// ---- FBs/Setpoint Optimizer/FB_SPOpt_HybridAirSystem.TcPOU
{attribute 'hide_all_locals'}
FUNCTION_BLOCK FB_SPOpt_HybridAirSystem
VAR_INPUT PERSISTENT
	bEnable							: BOOL;									//Enable or dissable thsi Function
END_VAR
VAR_INPUT
	byStateSystemIn					: BYTE;									//Actual State from the System. 0 = off, 1 = Heating mode on, 2 = Cooling Mode on
	rFlowAirTempIn					: REAL;									//Actual Flow Air Temperature
	rReturnAirTempIn				: REAL;									//Actual Return Air Temperature
	rInToOutAirTempIn				: REAL;									//Actual outdoor air flow temperature
	rOutToInAirTempIn				: REAL;									//Actual indoor air flow temperature
END_VAR
VAR_OUTPUT
	bError							: BOOL;									//Error from this Fuction
	byStateSystemOut				: BYTE;									//{#lynus.ag#()} //State from the System. 0 = off, 1 = Heating mode on, 2 = Cooling Mode on		
	rFlowAirTempOut					: REAL;									//{#lynus.ag#()} //Flow Air Temperature to send to the Backend Service.
	rReturnAirTempOut				: REAL;									//{#lynus.ag#()} //Return Air Temperature to send to the Backend Service.
	rInToOutAirTempOut				: REAL;									//{#lynus.ag#()} //Outdoor air flow temperature to send to the Backend Service.
	rOutToInAirTempOut				: REAL;									//{#lynus.ag#()} //Indoor air flow temperature to send to the Backend Service.
	diNrOfSPOpt_OUT					: DINT;									//Active Number from Setpoint Optimizer for using on other functions
END_VAR
VAR
	fbNumberDevice					: FB_NumberOfDevice;					//Function block to calcualte the number of the Device
	timDissableFunctions			: TON;									//Timer to dissable the Function after Lynus_Standards.Constants_General.tTimeDissableLynusFunctions Days without connection to the Lynus Cloud
	timResetConnectionOnGVL			: TON;									//Timer to try reset the connection Flag on the GVL. (When somebody delete the Connection Function and make only a onlinechange)
END_VAR

//Creator : Kai Ebensperger
//Company : Lynus AG
//Date : 03.12.2021
//Version : 1.0.0.0

//This Function is a Help Function for the Setpoint Optimizer on our Backend System
//Here we can read in the neccessary Values for a Hybrid Air System from a external Service and can send then to the Backend System for optimizing
//Hybrid System can bee heating and cooling
//Its Helpfull if we work with the TMC File

(*----------------------------------------------------------------------------------------Limits---------------------------------------------------------------------------------------------------------------*)

byStateSystemIn := LIMIT(0,byStateSystemIn,2);
	rFlowAirTempIn := LIMIT(-30,rFlowAirTempIn,150);
		rReturnAirTempIn := LIMIT(-30,rReturnAirTempIn,150);
			rInToOutAirTempIn := LIMIT(-30,rInToOutAirTempIn,150);
				rOutToInAirTempIn := LIMIT(-30,rOutToInAirTempIn,150);

(*-------------------------------------------------------------Calcualte the number of SP Opttimizer---------------------------------------------------------------*)

fbNumberDevice(
	diActualNumberOfDevices:= Lynus_Standards.GVL_Energy.stNumberOfDevices.diNumberOfSetPointOpt, 
	diMaxNumberOfDevices:= Constants_Energy.diMaxNumberOfSetPointOpt, 
	udiCounterOnlineChange:= TwinCAT_SystemInfoVarList._AppInfo.OnlineChangeCnt, 
	bNumberIsCalculatet=> , 
	bFPNumberIsCalculatet=> , 
	bOnlineChange=> , 
	diNumberForThisDevice=> diNrOfSPOpt_OUT, 
	diNumberOfTotalDevices=> );

//Write new Numer on GVL
IF fbNumberDevice.bFPNumberIsCalculatet THEN
	Lynus_Standards.GVL_Energy.stNumberOfDevices.diNumberOfSetPointOpt := fbNumberDevice.diNumberOfTotalDevices;	
END_IF 

//Delete old Number on GVL
IF fbNumberDevice.bOnlineChange THEN 
	Lynus_Standards.GVL_Energy.stNumberOfDevices.diNumberOfSetPointOpt := diNrOfSPOpt_OUT;
END_IF								
				
(*-------------------------------------------------------------Service from Backend is ready and check the connection to backen for dissabel/enable EMS Function---------------------------------------------------------------*)

//Try to reset the variable for connection on the GVL. When all is normal then the Lynus Mqtt connection function set this variable to true in the next cycle
//When we have no connection to the backend or no HB from the Service then after Lynus_Standards.Constants_General.tTimeDissableLynusFunctions days the EMS is dissabled with all of his functionalities
timResetConnectionOnGVL(IN:= NOT timResetConnectionOnGVL.Q, PT:= T#1H, Q=> , ET=> );
	IF timResetConnectionOnGVL.Q THEN Lynus_Standards.GVL_Communicator.bStateConnectionToEnableFunctions := FALSE; END_IF
		IF NOT Lynus_Standards.GVL_Communicator.bStateConnectionToEnableFunctions THEN timDissableFunctions.IN := TRUE; ELSE timDissableFunctions.IN := FALSE; END_IF  
			timDissableFunctions(IN:= , PT:= Lynus_Standards.Constants_General.tTimeDissableLynusFunctions, Q=> , ET=> );

(*------------------------------------------------------------------Error----------------------------------------------------------------------------*)	

IF Lynus_Standards.GVL_Energy.stNumberOfDevices.diNumberOfSetPointOpt > Constants_Energy.diMaxNumberOfSetPointOpt THEN bError := TRUE; ELSE bError := FALSE; END_IF 			
			
(*-------------------------------------------------------------------------------------In to Out---------------------------------------------------------------------------------------*)

byStateSystemOut := byStateSystemIn;
	rFlowAirTempOut := rFlowAirTempIn;
		rReturnAirTempOut := rReturnAirTempIn;	
			rInToOutAirTempOut := rInToOutAirTempIn;
				rOutToInAirTempOut := rOutToInAirTempIn;		

IF NOT bEnable OR timDissableFunctions.Q OR Lynus_Standards.GVL_Energy.stNumberOfDevices.diNumberOfSetPointOpt > Constants_Energy.diMaxNumberOfSetPointOpt THEN
	byStateSystemOut := 0;	
END_IF

END_FUNCTION_BLOCK

// ---- FBs/Setpoint Optimizer/FB_SPOpt_HybridWaterSystem.TcPOU
{attribute 'hide_all_locals'}
FUNCTION_BLOCK FB_SPOpt_HybridWaterSystem
VAR_INPUT PERSISTENT
	bEnable							: BOOL;									//Enable or dissable thsi Function
END_VAR
VAR_INPUT
	byStateSystemIn					: BYTE;									//Actual State from the System. 0 = off, 1 = Heating mode on, 2 = Cooling Mode on
	rFlowTempIn						: REAL;									//Actual Flow Temperature
	rReturnTempIn					: REAL;									//Actual Return Temperature
END_VAR
VAR_OUTPUT
	bError							: BOOL;									//Error from this Fuction
	byStateSystemOut				: BYTE;									//{#lynus.ag#()} //State from the System. 0 = off, 1 = Heating mode on, 2 = Cooling Mode on	
	rFlowTempOut					: REAL;									//{#lynus.ag#()} //Flow Temperature to send to the Backend Service.
	rReturnTempOut					: REAL;									//{#lynus.ag#()} //Return Temperature to send to the Backend Service.
	diNrOfSPOpt_OUT					: DINT;									//Active Number from Setpoint Optimizer for using on other functions
END_VAR
VAR
	fbNumberDevice					: FB_NumberOfDevice;					//Function block to calcualte the number of the Device
	timDissableFunctions			: TON;									//Timer to dissable the Function after Lynus_Standards.Constants_General.tTimeDissableLynusFunctions Days without connection to the Lynus Cloud
	timResetConnectionOnGVL			: TON;									//Timer to try reset the connection Flag on the GVL. (When somebody delete the Connection Function and make only a onlinechange)
END_VAR

//Creator : Kai Ebensperger
//Company : Lynus AG
//Date : 03.12.2021
//Version : 1.0.0.0

//This Function is a Help Function for the Setpoint Optimizer on our Backend System
//Here we can read in the neccessary Values for a Hybrid Water System from a external Service and can send then to the Backend System for optimizing
//Hybrid System can bee heating and cooling
//Its Helpfull if we work with the TMC File

(*----------------------------------------------------------------------------------------Limits---------------------------------------------------------------------------------------------------------------*)

byStateSystemIn := LIMIT(0,byStateSystemIn,2);
	rFlowTempIn := LIMIT(-30,rFlowTempIn,180);
		rReturnTempIn := LIMIT(-30,rReturnTempIn,180);

(*-------------------------------------------------------------Calcualte the number of SP Opttimizer---------------------------------------------------------------*)

fbNumberDevice(
	diActualNumberOfDevices:= Lynus_Standards.GVL_Energy.stNumberOfDevices.diNumberOfSetPointOpt, 
	diMaxNumberOfDevices:= Constants_Energy.diMaxNumberOfSetPointOpt, 
	udiCounterOnlineChange:= TwinCAT_SystemInfoVarList._AppInfo.OnlineChangeCnt, 
	bNumberIsCalculatet=> , 
	bFPNumberIsCalculatet=> , 
	bOnlineChange=> , 
	diNumberForThisDevice=> diNrOfSPOpt_OUT, 
	diNumberOfTotalDevices=> );

//Write new Numer on GVL
IF fbNumberDevice.bFPNumberIsCalculatet THEN
	Lynus_Standards.GVL_Energy.stNumberOfDevices.diNumberOfSetPointOpt := fbNumberDevice.diNumberOfTotalDevices;	
END_IF 

//Delete old Number on GVL
IF fbNumberDevice.bOnlineChange THEN 
	Lynus_Standards.GVL_Energy.stNumberOfDevices.diNumberOfSetPointOpt := diNrOfSPOpt_OUT;
END_IF			
		
(*-------------------------------------------------------------Service from Backend is ready and check the connection to backen for dissabel/enable EMS Function---------------------------------------------------------------*)

//Try to reset the variable for connection on the GVL. When all is normal then the Lynus Mqtt connection function set this variable to true in the next cycle
//When we have no connection to the backend or no HB from the Service then after Lynus_Standards.Constants_General.tTimeDissableLynusFunctions days the EMS is dissabled with all of his functionalities
timResetConnectionOnGVL(IN:= NOT timResetConnectionOnGVL.Q, PT:= T#1H, Q=> , ET=> );
	IF timResetConnectionOnGVL.Q THEN Lynus_Standards.GVL_Communicator.bStateConnectionToEnableFunctions := FALSE; END_IF
		IF NOT Lynus_Standards.GVL_Communicator.bStateConnectionToEnableFunctions THEN timDissableFunctions.IN := TRUE; ELSE timDissableFunctions.IN := FALSE; END_IF  
			timDissableFunctions(IN:= , PT:= Lynus_Standards.Constants_General.tTimeDissableLynusFunctions, Q=> , ET=> );

(*------------------------------------------------------------------Error----------------------------------------------------------------------------*)	

IF Lynus_Standards.GVL_Energy.stNumberOfDevices.diNumberOfSetPointOpt > Constants_Energy.diMaxNumberOfSetPointOpt THEN bError := TRUE; ELSE bError := FALSE; END_IF 			
			
(*-------------------------------------------------------------------------------------In to Out---------------------------------------------------------------------------------------*)

byStateSystemOut := byStateSystemIn;
	rFlowTempOut := rFlowTempIn;
		rReturnTempOut := rReturnTempIn;		

IF NOT bEnable OR timDissableFunctions.Q OR Lynus_Standards.GVL_Energy.stNumberOfDevices.diNumberOfSetPointOpt > Constants_Energy.diMaxNumberOfSetPointOpt THEN
	byStateSystemOut := 0;	
END_IF

END_FUNCTION_BLOCK

// ---- FBs/Setpoint Optimizer/FB_SPOpt_Monitoring.TcPOU
{attribute 'hide_all_locals'}
FUNCTION_BLOCK FB_SPOpt_Monitoring
VAR_INPUT PERSISTENT
	bEnable							: BOOL;									//{#lynus.ag#()} //Enable or dissable thsi function
	bDissableHB						: BOOL;									//If this is True, then the Output HB is also dissabled when we have a Error or the Ready Flag from the Backend Service is not OK. If its False the HB is only dissalbed when the Function is not Enables or the HB from the Backend Service is missing
	tChangeHBIn						: TIME := T#70S;						//Delay bettwen the changes from the HB at the Input HB Variable
	tChangeHBOut					: TIME := T#30S;						//Delay bettwen the changes from the HB at the Output HB Variable
END_VAR
VAR_INPUT
	rHeartbeat						: REAL;									//{#lynus.ag#()} //Heartbeat from the Service. NOT OVERRIDE
	rErrorWarning					: REAL;									//{#lynus.ag#()} //Error or Warning from the Service. NOT OVERRIDE
	rSPOptReady						: REAL;									//{#lynus.ag#()} //Setpoint Optimization Service Ready. NOT OVERRIDE
END_VAR
VAR_OUTPUT
	bError							: BOOL;									//Error from this Fuction
	bReadyOut						: BOOL;									//Show if the Service is Read or not
	bDissableExtHB					: BOOL;									//If someone use a external HB with this Flag he can see if the HB, ready or Error Flag from the Backend is set
	bSEnable						: BOOL;									//{#lynus.ag#()} //Enable State of hte function
	rHeartbeatOut					: REAL;									//Heartbeat for the external Service
	diNrOfSPOpt_OUT					: DINT;									//Active Number from Setpoint Optimizer for using on other functions
END_VAR
VAR
	rHBInput_CP						: REAL;									//Variable to compare input HB Variable to set or reset the timer
	fbNumberDevice					: FB_NumberOfDevice;					//Function block to calcualte the number of the Device
	timDissableFunctions			: TON;									//Timer to dissable the Function after Lynus_Standards.Constants_General.tTimeDissableLynusFunctions Days without connection to the Lynus Cloud
	timResetConnectionOnGVL			: TON;									//Timer to try reset the connection Flag on the GVL. (When somebody delete the Connection Function and make only a onlinechange)
	timHBInput						: TON;									//Timer to check the Input HB
	timHBOutput						: TON;									//Timer to set the Output HB
	timReady						: TON;									//Timer to dissable the Ready Flag
	timErrorWarning					: TON;									//Timmer do detect a Error or a Warning
END_VAR

//Creator : Kai Ebensperger
//Company : Lynus AG
//Date : 03.12.2021
//Version : 1.0.0.0

//This is a Function for using with the Setpoin Optimizer on our Backen System.
//So we have the possibility to send the Ready Flag and the HB to the external system we are communicating with in the right intervals.  
//Error evaluation also takes place in this function. Thus, in the event of an error or other event, the Ready flag, the HB or even both can be deactivated and the external system can switch back to classic control. 


(*-------------------------------------------------------------------------------Limits----------------------------------------------------------------------------------------------*)

rHeartbeat := LIMIT(0,rHeartbeat,1);
	rErrorWarning := LIMIT(0,rErrorWarning,2);
		rSPOptReady := LIMIT(0,rSPOptReady,1);
			tChangeHBIn := LIMIT(T#1S,tChangeHBIn,T#600S);
				tChangeHBOut := LIMIT(T#1S,tChangeHBOut,T#600S);	
	
(*-------------------------------------------------------------Calcualte the number of SP Opttimizer---------------------------------------------------------------*)

fbNumberDevice(
	diActualNumberOfDevices:= Lynus_Standards.GVL_Energy.stNumberOfDevices.diNumberOfSetPointOpt, 
	diMaxNumberOfDevices:= Constants_Energy.diMaxNumberOfSetPointOpt, 
	udiCounterOnlineChange:= TwinCAT_SystemInfoVarList._AppInfo.OnlineChangeCnt, 
	bNumberIsCalculatet=> , 
	bFPNumberIsCalculatet=> , 
	bOnlineChange=> , 
	diNumberForThisDevice=> diNrOfSPOpt_OUT, 
	diNumberOfTotalDevices=> );

//Write new Numer on GVL
IF fbNumberDevice.bFPNumberIsCalculatet THEN
	Lynus_Standards.GVL_Energy.stNumberOfDevices.diNumberOfSetPointOpt := fbNumberDevice.diNumberOfTotalDevices;	
END_IF 

//Delete old Number on GVL
IF fbNumberDevice.bOnlineChange THEN 
	Lynus_Standards.GVL_Energy.stNumberOfDevices.diNumberOfSetPointOpt := diNrOfSPOpt_OUT;
END_IF			
			
(*-------------------------------------------------------------Service from Backend is ready and check the connection to backen for dissabel/enable EMS Function---------------------------------------------------------------*)

//Try to reset the variable for connection on the GVL. When all is normal then the Lynus Mqtt connection function set this variable to true in the next cycle
//When we have no connection to the backend or no HB from the Service then after Lynus_Standards.Constants_General.tTimeDissableLynusFunctions days the EMS is dissabled with all of his functionalities
timResetConnectionOnGVL(IN:= NOT timResetConnectionOnGVL.Q, PT:= T#1H, Q=> , ET=> );
	IF timResetConnectionOnGVL.Q THEN Lynus_Standards.GVL_Communicator.bStateConnectionToEnableFunctions := FALSE; END_IF
		IF NOT Lynus_Standards.GVL_Communicator.bStateConnectionToEnableFunctions OR rHBInput_CP = rHeartbeat THEN timDissableFunctions.IN := TRUE; ELSE timDissableFunctions.IN := FALSE; END_IF  
			timDissableFunctions(IN:= , PT:= Lynus_Standards.Constants_General.tTimeDissableLynusFunctions, Q=> , ET=> );

(*------------------------------------------------------------------Error----------------------------------------------------------------------------*)	

IF Lynus_Standards.GVL_Energy.stNumberOfDevices.diNumberOfSetPointOpt > Constants_Energy.diMaxNumberOfSetPointOpt THEN bError := TRUE; ELSE bError := FALSE; END_IF 
			
(*-----------------------------------------------------------------------------------------------------Logic--------------------------------------------------------------------------------------------------------------*)

bSEnable := bEnable;

//Input HB
timHBInput(IN:= , PT:= tChangeHBIn, Q=> , ET=> );
	IF rHeartbeat <> rHBInput_CP THEN
		timHBInput.IN := FALSE; rHBInput_CP := rHeartbeat;
	ELSE
		timHBInput.IN := TRUE;
	END_IF

//Ready
IF rSPOptReady = 0 THEN timReady.IN := TRUE; ELSE timReady.IN := FALSE; END_IF
	timReady(IN:= , PT:= tChangeHBIn * 2, Q=> , ET=> ); 	
	
//Error and Warning
IF rErrorWarning <> 0 THEN timErrorWarning.IN := TRUE; ELSE timErrorWarning.IN := FALSE; END_IF
	timErrorWarning(IN:= , PT:= tChangeHBIn * 2, Q=> , ET=> );
	
//Set HB Output and Ready Flag
IF rSPOptReady <> 0 AND NOT timReady.Q AND bEnable AND NOT timDissableFunctions.Q AND NOT timErrorWarning.Q THEN bReadyOut := TRUE; END_IF
	IF timReady.Q OR timErrorWarning.Q THEN bReadyOut := FALSE; END_IF

IF (NOT timHBInput.Q AND bDissableHB AND bReadyOut AND NOT timErrorWarning.Q AND NOT timHBOutput.Q AND bEnable AND NOT timDissableFunctions.Q) OR
	(NOT timHBInput.Q AND NOT bDissableHB AND NOT timHBOutput.Q AND bEnable AND NOT timDissableFunctions.Q) THEN
		timHBOutput.IN := TRUE;
ELSE
		timHBOutput.IN := FALSE;
END_IF
	timHBOutput(IN:= , PT:= tChangeHBOut, Q=> , ET=> );
		IF timHBOutput.Q THEN rHeartbeatOut := rHeartbeatOut + 1; END_IF
 			IF rHeartbeatOut > 1 THEN rHeartbeatOut := 0; END_IF

//External HB Flag
IF timHBInput.Q OR (timReady.Q AND bDissableHB) OR (timErrorWarning.Q AND bDissableHB) THEN
	bDissableExtHB := TRUE;
ELSE
	bDissableExtHB := FALSE;
END_IF   
	
//Not Enabled
IF NOT bEnable OR timDissableFunctions.Q OR bError THEN
	bReadyOut := FALSE;
		bDissableExtHB := TRUE;
			rHeartbeatOut := 0;	
END_IF

END_FUNCTION_BLOCK

// ---- FBs/Setpoint Optimizer/FB_SPOpt_WaterSystem.TcPOU
{attribute 'hide_all_locals'}
FUNCTION_BLOCK FB_SPOpt_WaterSystem
VAR_INPUT PERSISTENT
	bEnable							: BOOL;									//Enable or dissable thsi Function
END_VAR
VAR_INPUT
	bExtCmdSysOnOff					: BOOL;									//{#lynus.ag#()} //External Command to swtich the system on or off. Use only for Heatign systems
	bErrorOutdoorTemp				: BOOL;									//Outdoor Temperatur Sensor has a Error
	byStateSystemIn					: BYTE;									//Actual State from the System. 0 = off, 1 = on
	rFlowTempIn						: REAL;									//Actual Flow Temperature
	rReturnTempIn					: REAL;									//Actual Return Temperature
	rActualOutdoorTemp				: REAL;									//Actual Outdoortemperature
END_VAR
VAR_OUTPUT
	bError							: BOOL;									//Error from this Fuction
	bExtCmdSysOnOffOut				: BOOL;									//Output to switch the System On or Off. Use only for Heatign systems
	byStateSystemOut				: BYTE;									//{#lynus.ag#()} //State from the System. 0 = off, 1 = on	
	rFlowTempOut					: REAL;									//{#lynus.ag#()} //Flow Temperature to send to the Backend Service.
	rReturnTempOut					: REAL;									//{#lynus.ag#()} //Return Temperature to send to the Backend Service.
	diNrOfSPOpt_OUT					: DINT;									//Active Number from Setpoint Optimizer for using on other functions
END_VAR
VAR
	fbNumberDevice					: FB_NumberOfDevice;					//Function block to calcualte the number of the Device
	timDissableFunctions			: TON;									//Timer to dissable the Function after Lynus_Standards.Constants_General.tTimeDissableLynusFunctions Days without connection to the Lynus Cloud
	timResetConnectionOnGVL			: TON;									//Timer to try reset the connection Flag on the GVL. (When somebody delete the Connection Function and make only a onlinechange)
END_VAR

//Creator : Kai Ebensperger
//Company : Lynus AG
//Date : 03.12.2021
//Version : 1.0.0.0

//This Function is a Help Function for the Setpoint Optimizer on our Backend System
//Here we can read in the neccessary Values for a Water System from a external Service and can send then to the Backend System for optimizing
//Its Helpfull if we work with the TMC File

(*----------------------------------------------------------------------------------------Limits---------------------------------------------------------------------------------------------------------------*)

byStateSystemIn := LIMIT(0,byStateSystemIn,1);
	rFlowTempIn := LIMIT(-30,rFlowTempIn,180);
		rReturnTempIn := LIMIT(-30,rReturnTempIn,180);

(*-------------------------------------------------------------Calcualte the number of SP Opttimizer---------------------------------------------------------------*)

fbNumberDevice(
	diActualNumberOfDevices:= Lynus_Standards.GVL_Energy.stNumberOfDevices.diNumberOfSetPointOpt, 
	diMaxNumberOfDevices:= Constants_Energy.diMaxNumberOfSetPointOpt, 
	udiCounterOnlineChange:= TwinCAT_SystemInfoVarList._AppInfo.OnlineChangeCnt, 
	bNumberIsCalculatet=> , 
	bFPNumberIsCalculatet=> , 
	bOnlineChange=> , 
	diNumberForThisDevice=> diNrOfSPOpt_OUT, 
	diNumberOfTotalDevices=> );

//Write new Numer on GVL
IF fbNumberDevice.bFPNumberIsCalculatet THEN
	Lynus_Standards.GVL_Energy.stNumberOfDevices.diNumberOfSetPointOpt := fbNumberDevice.diNumberOfTotalDevices;	
END_IF 

//Delete old Number on GVL
IF fbNumberDevice.bOnlineChange THEN 
	Lynus_Standards.GVL_Energy.stNumberOfDevices.diNumberOfSetPointOpt := diNrOfSPOpt_OUT;
END_IF			
		
(*-------------------------------------------------------------Service from Backend is ready and check the connection to backen for dissabel/enable EMS Function---------------------------------------------------------------*)

//Try to reset the variable for connection on the GVL. When all is normal then the Lynus Mqtt connection function set this variable to true in the next cycle
//When we have no connection to the backend or no HB from the Service then after Lynus_Standards.Constants_General.tTimeDissableLynusFunctions days the EMS is dissabled with all of his functionalities
timResetConnectionOnGVL(IN:= NOT timResetConnectionOnGVL.Q, PT:= T#1H, Q=> , ET=> );
	IF timResetConnectionOnGVL.Q THEN Lynus_Standards.GVL_Communicator.bStateConnectionToEnableFunctions := FALSE; END_IF
		IF NOT Lynus_Standards.GVL_Communicator.bStateConnectionToEnableFunctions THEN timDissableFunctions.IN := TRUE; ELSE timDissableFunctions.IN := FALSE; END_IF  
			timDissableFunctions(IN:= , PT:= Lynus_Standards.Constants_General.tTimeDissableLynusFunctions, Q=> , ET=> );

(*------------------------------------------------------------------Error----------------------------------------------------------------------------*)	

IF Lynus_Standards.GVL_Energy.stNumberOfDevices.diNumberOfSetPointOpt > Constants_Energy.diMaxNumberOfSetPointOpt THEN bError := TRUE; ELSE bError := FALSE; END_IF 			
			
(*-------------------------------------------------------------------------------------In to Out---------------------------------------------------------------------------------------*)

byStateSystemOut := byStateSystemIn;
	rFlowTempOut := rFlowTempIn;
		rReturnTempOut := rReturnTempIn;		

IF NOT bEnable OR timDissableFunctions.Q OR Lynus_Standards.GVL_Energy.stNumberOfDevices.diNumberOfSetPointOpt > Constants_Energy.diMaxNumberOfSetPointOpt THEN
	byStateSystemOut := 0;	
END_IF

(*-------------------------------------------------------------------------------------External On/Off Command---------------------------------------------------------------------------------------*)

//On
bExtCmdSysOnOffOut := TRUE;
	//Off
	IF NOT bExtCmdSysOnOff AND rActualOutdoorTemp > 5 AND NOT bErrorOutdoorTemp THEN bExtCmdSysOnOffOut := FALSE; END_IF

END_FUNCTION_BLOCK

// ---- FBs/Valve Control/OnOff/FB_Valve_Control_MPC_HCO_DO.TcPOU
FUNCTION_BLOCK FB_Valve_Control_MPC_HCO_DO
VAR_INPUT PERSISTENT
	bEnable								: BOOL;												//Enable or dissable the function
	diNrOfTempS_IN_FlowTemp				: DINT;												//Number of the Temperature Sensor for incoming temperature data. (Temperature Sensor for the Flow Temperature)
	diNrOfTempS_IN_ReturnTemp			: DINT;												//Number of the Temperature Sensor for incoming temperature data. (Temperature Sensor for the Return Temperature)
	diNrOfTempS_IN_RoomTemp				: DINT;												//Number of the Temperature Sensor for incoming temperature data. (Temperature Sensor for the Room Temperature)
END_VAR
VAR_OUTPUT
	stDataValveControlOut				: ST_Valve_Control_Output;							//{#lynus.ag#()} //Valve Control output data
	byErrorWarning						: BYTE;												//{#lynus.ag#()} //Shows the Error and Warning State from the Backend Service
	byMPCReady							: BYTE;												//{#lynus.ag#()} //Shows if the MPC service is ready or not.
	byNewValvePosition					: BYTE;												//{#lynus.ag#()} //The new valve positon from the Lynus Backend Service
	diNrOfValveControl_OUT				: DINT;												//Active Number from the Valve Controling for using on other functions
	rFlowTemperatureRoom				: REAL;												//{#lynus.ag#()} //Shows the actual Flow temperature from the Heating Circuit
	rReturnTemperatureRoom				: REAL;												//{#lynus.ag#()} //Shows the actual Return temperature from the Heating Circuit
	rActualRoomTemperature				: REAL;												//{#lynus.ag#()} //Shows the actual Room temperature
	rNewRoomTemperature					: REAL;												//{#lynus.ag#()} //Shows the new Room Temperture for the next hour
	rHeartbeat							: REAL;												//{#lynus.ag#()} //Heartbeat from the Backend Service
	rNewSetTemperature					: REAL;												//{#lynus.ag#()} //New Set Temperatur on witch the Valve is switching on and off
END_VAR
VAR
	{attribute 'hide'}
	fbValveControl						: FB_Valve_Control;									//Function for Valve controll
	{attribute 'hide'}
	fbNumberDevice						: FB_NumberOfDevice;								//Function block to calcualte the number of the Device
	fbDOOnOffValve						: FB_XL2XXX_DO;										//Digital Output to swtich the valve on and off
	{attribute 'hide'}
	timDissableFunctions				: TON;												//Timer to dissable the Function after Lynus_Standards.Constants_General.tTimeDissableLynusFunctions Days without connection to the Lynus Cloud
	{attribute 'hide'}
	timResetConnectionOnGVL				: TON;												//Timer to try reset the connection Flag on the GVL. (When somebody delete the Connection Function and make only a onlinechange)
	{attribute 'hide'}
	arrPD								: ARRAY[1..4] OF FB_PersistentData_Number;			//Function to save persistent data 
	{attribute 'hide'}
	byWaitInStep						: BYTE;												//Wait in Step before start to clean data on PLC
	{attribute 'hide'}
	iStateGVLData						: INT;												//State machine to handle the data on the GVL
	{attribute 'hide'}
	diCounterForGVL						: DINT;												//Counter to clean old data on GVL
END_VAR

//Creator : Kai Ebensperger
//Company : Lynus AG
//Date : 21.07.2021
//Version : 1.0.0.0

//With this function its possible to control a floor heating valve or radiator valve.
//The signal is sending to a digital output terminal.
//The Backend is connected with this Function to optimize the regulation of the valve 

//NOTE for diNr.....Designation => 
//_IN = Here Data come in from other Functions or go out to other functions about the GVL
//_OUT = Here Data go out to other functions about the GVL

(*------------------------------------------------------------Limits----------------------------------------------------------------------------------*)

diNrOfTempS_IN_FlowTemp := LIMIT(0,diNrOfTempS_IN_FlowTemp,Constants_Sensors.diMaxNumberOfTemperatureSensors);
	diNrOfTempS_IN_ReturnTemp := LIMIT(0,diNrOfTempS_IN_ReturnTemp,Constants_Sensors.diMaxNumberOfTemperatureSensors);
		diNrOfTempS_IN_RoomTemp := LIMIT(0,diNrOfTempS_IN_RoomTemp,Constants_Sensors.diMaxNumberOfTemperatureSensors);

(*-------------------------------------------------------------Calcualte the number of valve control---------------------------------------------------------------*)

fbNumberDevice(
	diActualNumberOfDevices:= Lynus_Standards.GVL_Energy.stNumberOfDevices.diNumberOfValveControls, 
	diMaxNumberOfDevices:= Constants_Energy.diMaxNumberOfValveControls, 
	udiCounterOnlineChange:= TwinCAT_SystemInfoVarList._AppInfo.OnlineChangeCnt, 
	bNumberIsCalculatet=> , 
	bFPNumberIsCalculatet=> , 
	bOnlineChange=> , 
	diNumberForThisDevice=> diNrOfValveControl_OUT, 
	diNumberOfTotalDevices=> );

//Write new Numer on GVL
IF fbNumberDevice.bFPNumberIsCalculatet THEN
	Lynus_Standards.GVL_Energy.stNumberOfDevices.diNumberOfValveControls := fbNumberDevice.diNumberOfTotalDevices;	
END_IF 

//Delete old Number on GVL
IF fbNumberDevice.bOnlineChange THEN 
	Lynus_Standards.GVL_Energy.stNumberOfDevices.diNumberOfValveControls := diNrOfValveControl_OUT;	
		iStateGVLData := 1; 
END_IF

(*-------------------------------------------------------------Service from Backend is ready and check the connection to backen for dissabel/enable Function---------------------------------------------------------------*)

//Try to reset the variable for connection on the GVL. When all is normal then the Lynus Mqtt connection function set this variable to true in the next cycle
//When we have no connection to the backend then after Lynus_Standards.Constants_General.tTimeDissableLynusFunctions days the Function is dissabled with all of his functionalities
timResetConnectionOnGVL(IN:= NOT timResetConnectionOnGVL.Q, PT:= T#1H, Q=> , ET=> );
	IF timResetConnectionOnGVL.Q THEN Lynus_Standards.GVL_Communicator.bStateConnectionToEnableFunctions := FALSE; END_IF
		IF NOT Lynus_Standards.GVL_Communicator.bStateConnectionToEnableFunctions THEN timDissableFunctions.IN := TRUE; ELSE timDissableFunctions.IN := FALSE; END_IF  
			timDissableFunctions(IN:= , PT:= Lynus_Standards.Constants_General.tTimeDissableLynusFunctions, Q=> , ET=> );

(*------------------------------------------------------------------Error-Warning----------------------------------------------------------------------------*)				
			
IF timDissableFunctions.Q OR byErrorWarning = 1 THEN fbValveControl.bWarning := TRUE; ELSE fbValveControl.bWarning := FALSE; END_IF 	
	IF Lynus_Standards.GVL_Energy.stNumberOfDevices.diNumberOfValveControls > Constants_Energy.diMaxNumberOfValveControls OR byErrorWarning = 2 OR 
		(Lynus_Standards.GVL_Sensors.stDataTemperatureSensors[diNrOfTempS_IN_FlowTemp].bEnabled AND Lynus_Standards.GVL_Sensors.stDataTemperatureSensors[diNrOfTempS_IN_FlowTemp].byErrorWarning = 2) OR	
			(Lynus_Standards.GVL_Sensors.stDataTemperatureSensors[diNrOfTempS_IN_ReturnTemp].bEnabled AND Lynus_Standards.GVL_Sensors.stDataTemperatureSensors[diNrOfTempS_IN_ReturnTemp].byErrorWarning = 2) OR	
				(Lynus_Standards.GVL_Sensors.stDataTemperatureSensors[diNrOfTempS_IN_RoomTemp].bEnabled AND Lynus_Standards.GVL_Sensors.stDataTemperatureSensors[diNrOfTempS_IN_RoomTemp].byErrorWarning = 2) THEN
					fbValveControl.bError := TRUE; 
	ELSE 
					fbValveControl.bError := FALSE; 
	END_IF 
		//Warning Codes
		IF byErrorWarning = 1 THEN fbValveControl.iWarningCode := 1;
		ELSIF timDissableFunctions.Q THEN fbValveControl.iWarningCode := 0;
		END_IF
		//Error Code
		IF byErrorWarning = 2 THEN fbValveControl.iErrorCode := 2;
		ELSIF Lynus_Standards.GVL_Sensors.stDataTemperatureSensors[diNrOfTempS_IN_FlowTemp].bEnabled AND Lynus_Standards.GVL_Sensors.stDataTemperatureSensors[diNrOfTempS_IN_FlowTemp].byErrorWarning = 2 THEN fbValveControl.iErrorCode := 3;
		ELSIF Lynus_Standards.GVL_Sensors.stDataTemperatureSensors[diNrOfTempS_IN_ReturnTemp].bEnabled AND Lynus_Standards.GVL_Sensors.stDataTemperatureSensors[diNrOfTempS_IN_ReturnTemp].byErrorWarning = 2 THEN fbValveControl.iErrorCode := 3;
		ELSIF Lynus_Standards.GVL_Sensors.stDataTemperatureSensors[diNrOfTempS_IN_RoomTemp].bEnabled AND Lynus_Standards.GVL_Sensors.stDataTemperatureSensors[diNrOfTempS_IN_RoomTemp].byErrorWarning = 2 THEN fbValveControl.iErrorCode := 3; 	
		ELSIF Lynus_Standards.GVL_Energy.stNumberOfDevices.diNumberOfValveControls > Constants_Energy.diMaxNumberOfValveControls THEN fbValveControl.iErrorCode := 1;
		END_IF   
		
fbValveControl(
	bEnable:= bEnable AND NOT timDissableFunctions.Q, 
	bWriteWithDelay:= TRUE, 
	bWorkOnlyLocal:= FALSE, 
	rActualRoomTemperature:= Lynus_Standards.GVL_Sensors.stDataTemperatureSensors[diNrOfTempS_IN_RoomTemp].rTemperature, 
	bError:= , 
	bWarning:= , 
	iErrorCode:= , 
	iWarningCode:= , 
	tTimDelayOutput:= T#5S, 
	byMPCReady:= byMPCReady, 
	byNewValvePosition:= byNewValvePosition, 
	rNewSetTemperature:= rNewSetTemperature, 
	rHeartbeat:= rHeartbeat, 
	stDataValveControlOut=> , 
	stDataValveControlOutDelay=> stDataValveControlOut);
	
(*-------------------------------------------------------------------------Output----------------------------------------------------------------------*)

//Send this data to the cloud service
rFlowTemperatureRoom := Lynus_Standards.GVL_Sensors.stDataTemperatureSensors[diNrOfTempS_IN_FlowTemp].rTemperature;
	rReturnTemperatureRoom := Lynus_Standards.GVL_Sensors.stDataTemperatureSensors[diNrOfTempS_IN_ReturnTemp].rTemperature;
		rActualRoomTemperature := Lynus_Standards.GVL_Sensors.stDataTemperatureSensors[diNrOfTempS_IN_RoomTemp].rTemperature; 

//Send the valve signal to the Digital output
fbDOOnOffValve(bInvers:= FALSE, bSignal:= fbValveControl.stDataValveControlOut.bValvePos);	

(*-----------------------------------------------------------Handle data to Global structure for the valve controling-----------------------------------------------------------------*)

CASE iStateGVLData OF
	
	0://Init Step
		byWaitInStep := 0;
			diCounterForGVL := 1;
	
	1://Wait for 4 Steps before clean al Data on GVL
		byWaitInStep := byWaitInStep + 1;
			IF byWaitInStep >= 4 AND fbNumberDevice.bNumberIsCalculatet THEN iStateGVLData := 2; END_IF
				//To much Devices, back to the Init step
				IF byWaitInStep >= 4 AND NOT fbNumberDevice.bNumberIsCalculatet THEN iStateGVLData := 0; END_IF	
			
	2://Clear all Data in GVL
		Lynus_Standards.GVL_Energy.stDataValveControls[diCounterForGVL].bEnabled := FALSE;
			Lynus_Standards.GVL_Energy.stDataValveControls[diCounterForGVL].byErrorWarning := 0;
				Lynus_Standards.GVL_Energy.stDataValveControls[diCounterForGVL].bValvePos := FALSE;
		
		diCounterForGVL := diCounterForGVL + 1;
			diCounterForGVL := LIMIT(0,diCounterForGVL,Constants_Energy.diMaxNumberOfValveControls);
				//Back to the init step
				IF diCounterForGVL >= Constants_Energy.diMaxNumberOfValveControls THEN iStateGVLData := 0; END_IF

END_CASE 	 

IF diNrOfValveControl_OUT > 0 AND fbNumberDevice.bNumberIsCalculatet THEN
	Lynus_Standards.GVL_Energy.stDataValveControls[diNrOfValveControl_OUT].bEnabled := fbValveControl.stDataValveControlOut.bEnabled;
		Lynus_Standards.GVL_Energy.stDataValveControls[diNrOfValveControl_OUT].byErrorWarning := fbValveControl.stDataValveControlOut.byErrorWarning;
			Lynus_Standards.GVL_Energy.stDataValveControls[diNrOfValveControl_OUT].bValvePos := fbValveControl.stDataValveControlOut.bValvePos;
END_IF

(*----------------------------------------------------------Save persistent data----------------------------------------------------------------*)

arrPD[1](lrValue:= BOOL_TO_LREAL(bEnable), bEventBasedActive=> );
arrPD[2](lrValue:= DINT_TO_LREAL(diNrOfTempS_IN_FlowTemp), bEventBasedActive=> );
arrPD[3](lrValue:= DINT_TO_LREAL(diNrOfTempS_IN_ReturnTemp), bEventBasedActive=> );
arrPD[4](lrValue:= DINT_TO_LREAL(diNrOfTempS_IN_RoomTemp), bEventBasedActive=> );

END_FUNCTION_BLOCK
